// TIA Portal V20 export
VAR_GLOBAL   // PLC tag table "Cabinet_5_6"
   Sz5_ST01_SenA AT %I1504.0 : Bool;
   Sz5_ST01_SenB AT %I1504.1 : Bool;
   Sz5_ST01_SenC AT %I1504.2 : Bool;
   Sz5_ST01_SenD AT %I1504.3 : Bool;
   Sz5_ST02_SenA AT %I1504.4 : Bool;
   Sz5_ST02_SenB AT %I1504.5 : Bool;
   Sz5_ST02_SenC AT %I1504.6 : Bool;
   Sz5_ST02_SenD AT %I1504.7 : Bool;
   Sz5_ST34_SenA AT %I1505.0 : Bool;
   Sz5_ST34_SenB AT %I1505.1 : Bool;
   Sz5_ST34_SenC AT %I1505.2 : Bool;
   Sz5_ST34_SenD AT %I1505.3 : Bool;
   Sz5_ST35_SenA AT %I1505.4 : Bool;
   Sz5_ST35_SenB AT %I1505.5 : Bool;
   Sz5_ST35_SenC AT %I1505.6 : Bool;
   Sz5_ST35_SenD AT %I1505.7 : Bool;
   Sz5_ST38_SenA AT %I1506.0 : Bool;
   Sz5_ST38_SenB AT %I1506.1 : Bool;
   Sz5_ST38_SenC AT %I1506.2 : Bool;
   Sz5_ST38_SenD AT %I1506.3 : Bool;
   Arm1_LowerClampOpen AT %I1500.0 : Bool;
   Arm1_LowerClampClosed AT %I1500.1 : Bool;
   Arm1_UpperClampOpen AT %I1500.2 : Bool;
   Arm1_UpperClampClosed AT %I1500.3 : Bool;
   Arm2_LowerClampOpen AT %I1500.4 : Bool;
   Arm2_UpperClampOpen AT %I1500.5 : Bool;
   Arm2_LowerClampClosed AT %I1500.6 : Bool;
   Arm2_UpperClampClosed AT %I1500.7 : Bool;
   S5_Arm1_BasePos AT %I1501.0 : Bool;
   S5_Arm2_BasePos AT %I1501.1 : Bool;
   S5_HydraulicStatus AT %I1501.2 : Bool;
   Arm1_Inclinometer AT %I1507.0 : "PII - JN2200";
   Arm2_Inclinometer AT %I1513.0 : "PII - JN2200";
   S6_Button_Up AT %I1501.5 : Bool;
   S5_Button_ST01_ST02 AT %I1502.0 : Bool;
   S5_Button_ST02_ST01 AT %I1502.1 : Bool;
   S5_Button_ST34_ST35 AT %I1502.2 : Bool;
   S5_Button_ST35_ST34 AT %I1502.3 : Bool;
   S5_Button_ST38_ST01 AT %I1502.4 : Bool;
   S5_Button_ST01_ST38 AT %I1502.5 : Bool;
   S5_Button_ST35 AT %I1502.6 : Bool;
   S5_Button_ST02 AT %I1502.7 : Bool;
   S5_Button_ST03 AT %I1503.0 : Bool;
   S5_Button_ST04 AT %I1503.1 : Bool;
   S5_Button_SS1_Up AT %I1503.2 : Bool;
   S5_Button_SS1_Down AT %I1503.3 : Bool;
   S5_Button_Buzz AT %I1503.4 : Bool;
   S6_Button_Buzz AT %I1503.5 : Bool;
   S5_Button_down AT %I1503.6 : Bool;
   Sz5_Estop_chA AT %I1550.0 : Bool;
   Sz6_Estop_chA AT %I1550.1 : Bool;
   Sz5_Estop_chB AT %I1550.3 : Bool;
   Sz6_Estop_chB AT %I1550.4 : Bool;
   TipHydSoftstart AT %Q2101.0 : Bool;
   TipHydContactor AT %Q2101.1 : Bool;
   UpperClampsClose AT %Q1500.0 : Bool;
   UpperClampsOpen AT %Q1500.1 : Bool;
   LowerClampsOpen AT %Q1500.2 : Bool;
   LowerClampsClose AT %Q1500.3 : Bool;
   S5_Button_LED_ST01_ST02 AT %Q1501.0 : Bool;
   S5_Button_LED_ST02_ST01 AT %Q1501.1 : Bool;
   S5_Button_LED_ST34_ST35 AT %Q1501.2 : Bool;
   S5_Button_LED_ST35_ST34 AT %Q1501.3 : Bool;
   S5_Button_LED_ST38_ST01 AT %Q1501.4 : Bool;
   S5_Button_LED_ST01_ST38 AT %Q1501.5 : Bool;
   S5_Button_LED_ST35 AT %Q1501.6 : Bool;
   S5_Button_LED_ST02 AT %Q1501.7 : Bool;
   S5_Button_LED_ST03 AT %Q1502.0 : Bool;
   S5_Button_LED_ST04 AT %Q1502.1 : Bool;
   S5_Button_LED_SS1_Up AT %Q1502.2 : Bool;
   S5_Button_LED_SS1_Down AT %Q1502.3 : Bool;
   S5_Button_LED_Buzz AT %Q1502.4 : Bool;
   S6_Button_LED_Up AT %Q1502.5 : Bool;
   S6_Button_LED_Buzz AT %Q1502.6 : Bool;
   S5_Button_LED_Down AT %Q1502.7 : Bool;
   TipArm1 AT %QW1542 : Int;
   TipArm2 AT %QW1544 : Int;
END_VAR
